TYPE general_input_datagrid_params :
STRUCT
	tension : LREAL;
	linspeed : LREAL;
	unwinding : BOOL;
END_STRUCT
END_TYPE

(* stored: Version 1.1.0.1, ProductVersion 3.1.4024.12
   DUT general_input_datagrid_params: Id {bde90c17-6b58-4868-83e2-051b3b1f7058} *)
